FUNCTION_BLOCK FBGenerateData
VAR_IN_OUT
	data : ST_SensorData;
END_VAR

VAR
	rand : drand;
	value: LREAL;
END_VAR

rand(Seed:=LREAL_TO_INT(value));
value := rand.Num;
data.rSensorValue := LREAL_TO_REAL(value);

END_FUNCTION_BLOCK

(* stored: Version 1.1.0.1, ProductVersion 3.1.4024.9
   POU FBGenerateData: Id {42f30776-c234-4b5b-8e0e-3250c8f558c1}, SpecialFunc None *)
